Fanuc KAREL source: GET_JPOS_REG.kl

PROGRAM T
%NOLOCKGROUP
VAR
 v0 : INTEGER
 v1 : INTEGER
 v2 : INTEGER
 res : JOINTPOS
BEGIN
 res = GET_JPOS_REG(v0, v1, v2)
END T
